// TIA Portal V20 export
FUNCTION "TIC100" : Void   // FC22, FBD
{ S7_Optimized_Access := 'TRUE' }
// stored: SetENOAutomatically false
   VAR_TEMP
      Temp : "DigVal";
      TempSP_Raw : Real;
      Temp_TimeMs : DInt;
      Temp_TimeSec : DInt;
      SP_Ext : "AnaVal";
      State : "Service_States";
      ChIn_PVOut : "AnaVal";
      TIC_PV : "AnaVal";
   END_VAR
BEGIN

REGION Network 1: Channel input
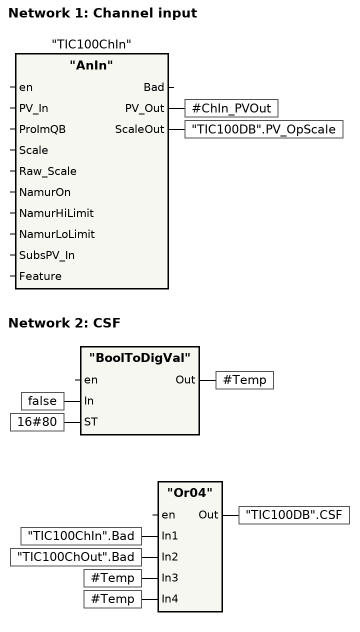
   "TIC100ChIn"(PV_Out => #ChIn_PVOut, ScaleOut => "TIC100DB".PV_OpScale);   // "AnIn"
END_REGION

REGION Network 2: CSF
   "BoolToDigVal"(In := false, ST := 16#80, Out => #Temp);
   "Or04"(In1 := "TIC100ChIn".Bad, In2 := "TIC100ChOut".Bad, In3 := #Temp, In4 := #Temp, Out => "TIC100DB".CSF);
END_REGION

REGION Network 3: Interlock
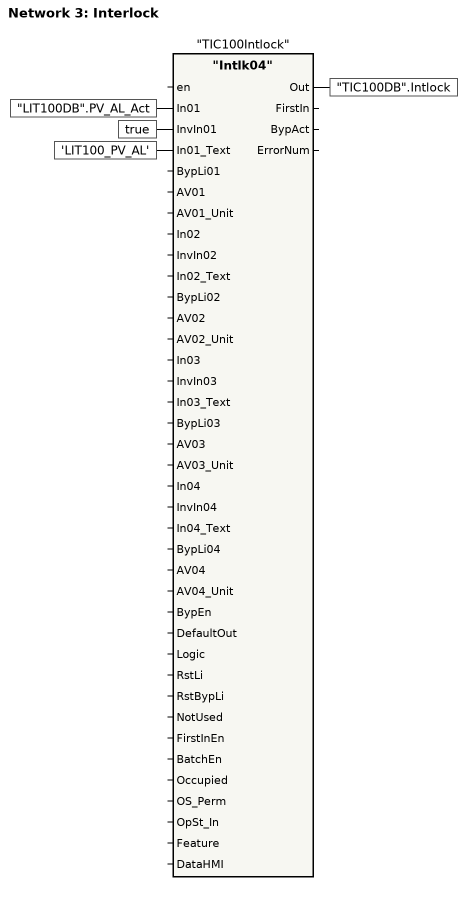
   "TIC100Intlock"(In01 := "LIT100DB".PV_AL_Act,   // "Intlk04"
                   InvIn01 := true,
                   In01_Text := 'LIT100_PV_AL',
                   Out => "TIC100DB".Intlock);
END_REGION

REGION Network 4: PIDCon
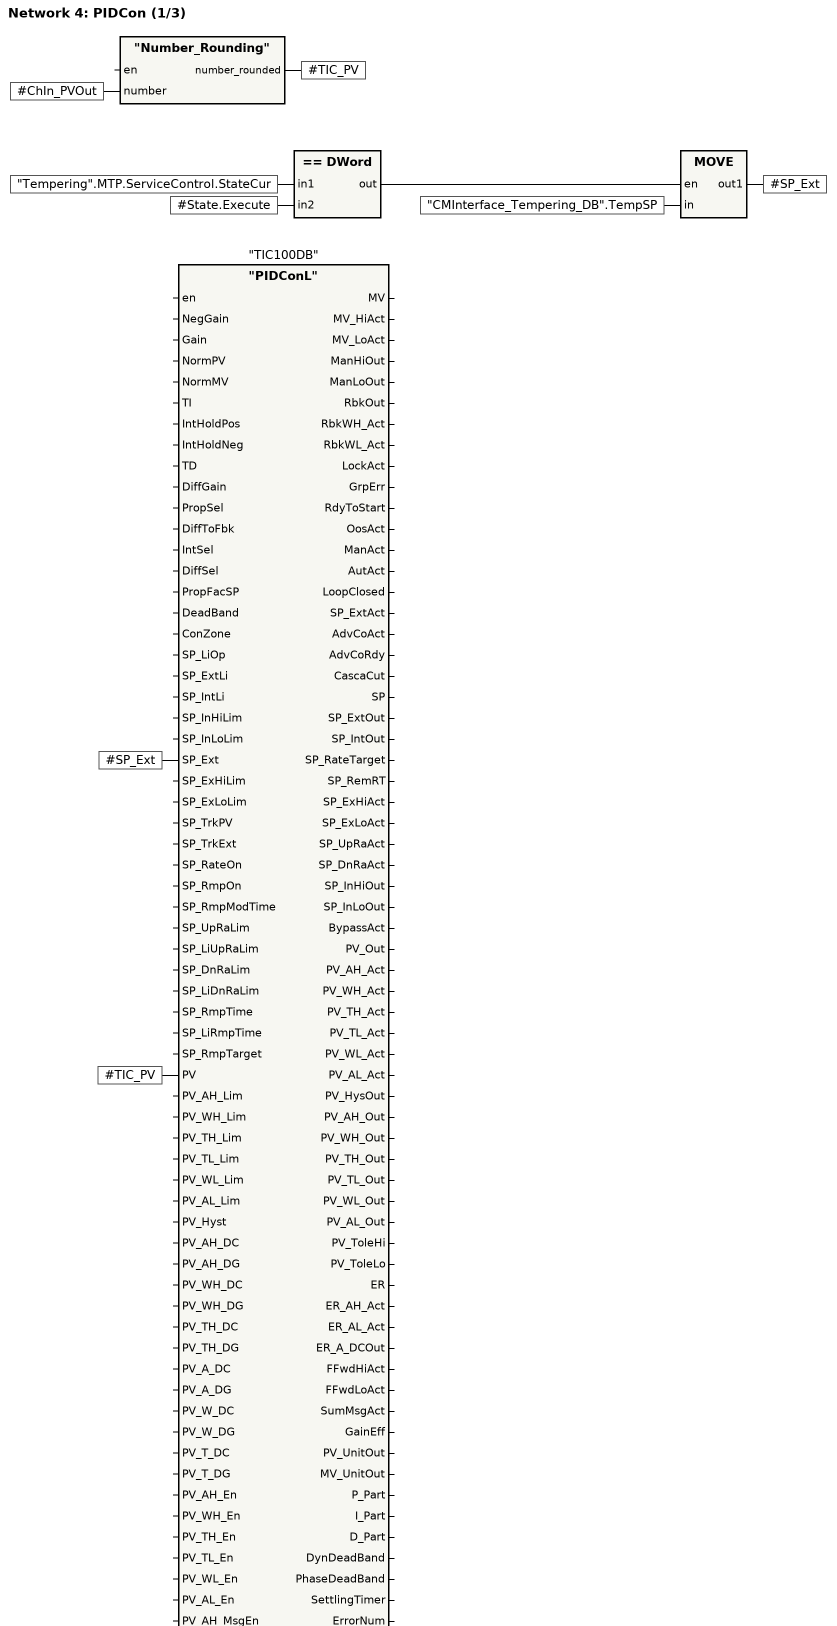
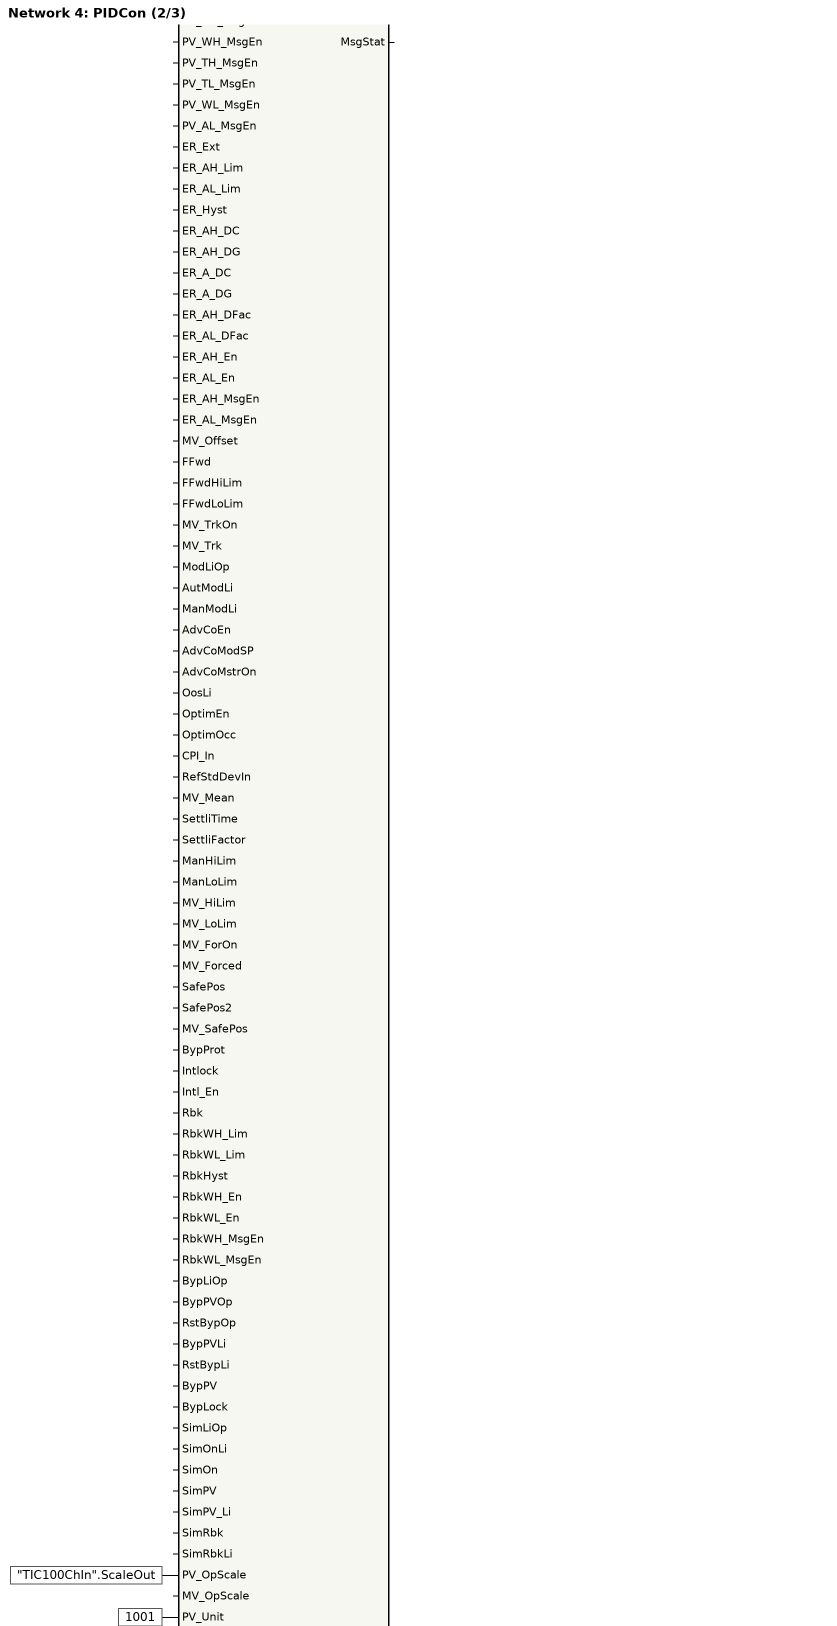
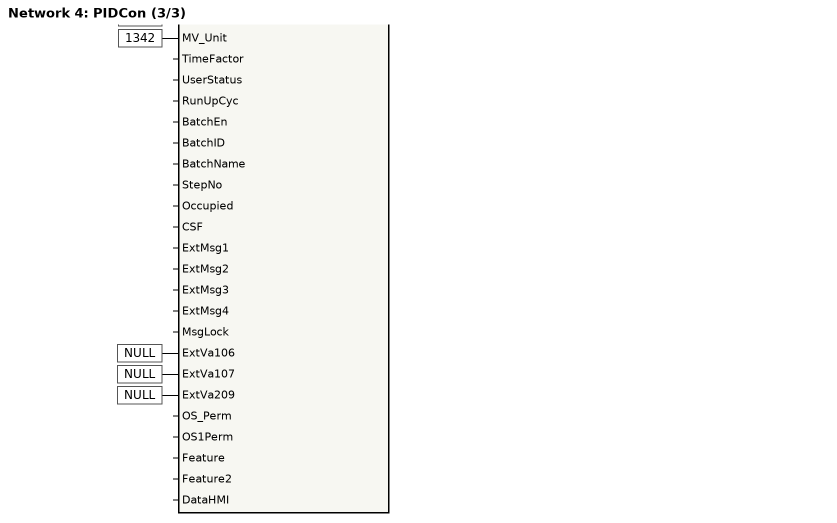
   "Number_Rounding"(number := #ChIn_PVOut, number_rounded => #TIC_PV);
   IF "Tempering".MTP.ServiceControl.StateCur = #State.Execute THEN
       #SP_Ext := "CMInterface_Tempering_DB".TempSP;
   END_IF;
   "TIC100DB"(SP_Ext := #SP_Ext,   // "PIDConL"
              PV := #TIC_PV,
              PV_OpScale := "TIC100ChIn".ScaleOut,
              PV_Unit := 1001,
              MV_Unit := 1342,
              ExtVa106 := NULL,
              ExtVa107 := NULL,
              ExtVa209 := NULL);
END_REGION

REGION Network 5: MTP
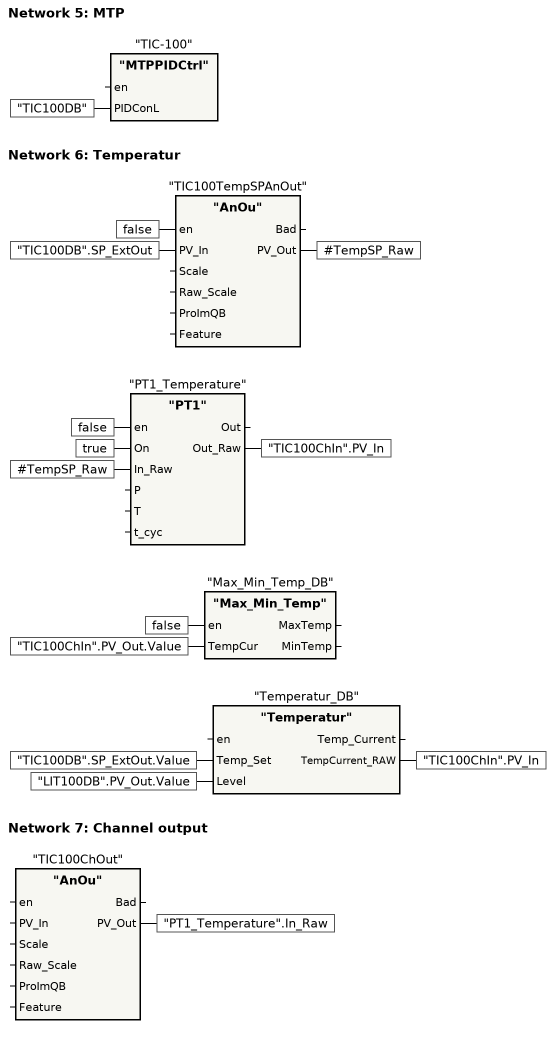
   "TIC-100"(PIDConL := "TIC100DB");   // "MTPPIDCtrl"
END_REGION

REGION Network 6: Temperatur
   IF false THEN
       "TIC100TempSPAnOut"(PV_In := "TIC100DB".SP_ExtOut, PV_Out => #TempSP_Raw);   // "AnOu"
       "PT1_Temperature"(On := true, In_Raw := #TempSP_Raw, Out_Raw => "TIC100ChIn".PV_In);   // "PT1"
       "Max_Min_Temp_DB"(TempCur := "TIC100ChIn".PV_Out.Value);   // "Max_Min_Temp"
   END_IF;
   "Temperatur_DB"(Temp_Set := "TIC100DB".SP_ExtOut.Value,   // "Temperatur"
                   Level := "LIT100DB".PV_Out.Value,
                   TempCurrent_RAW => "TIC100ChIn".PV_In);
END_REGION

REGION Network 7: Channel output
   "TIC100ChOut"(PV_Out => "PT1_Temperature".In_Raw);   // "AnOu"
END_REGION
END_FUNCTION
